INTERFACE I_DWORD EXTENDS I_Datatype

PROPERTY PUBLIC Value : REFERENCE TO DWORD
GET
END_GET
END_PROPERTY

END_INTERFACE

(* stored: Version 1.1.0.1, ProductVersion 3.1.4024.15
   Itf I_DWORD: Id {c9761be7-68dc-0017-2913-62a6ff111009}
   Property Value: Id {4bde9af6-d2d3-093b-2f88-f4ae90fc92c4}
   Get Get: Id {2570573c-3036-01d9-266a-a7015d8d1794} *)
